FUNCTION_BLOCK OutputPipe (* Composite Function Block Type *)
  (* Standard: 61499-2 *)
  (* Version 0.0, 2011-12-23, 4DIAC-IDE, 4DIAC-Consortium *)
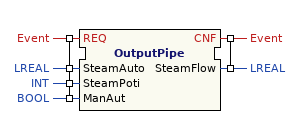
  EVENT_INPUT
    REQ WITH SteamAuto, SteamPoti, ManAut; (* Normal Execution Request *)
  END_EVENT
  EVENT_OUTPUT
    CNF WITH SteamFlow; (* Execution Confirmation *)
  END_EVENT
  VAR_INPUT
    SteamAuto : LREAL; (* Input event qualifier *)
    SteamPoti : INT;
    ManAut : BOOL; (* 0:Man, 1:Auto *)
  END_VAR
  VAR_OUTPUT
    SteamFlow : LREAL; (* Output event qualifier *)
  END_VAR
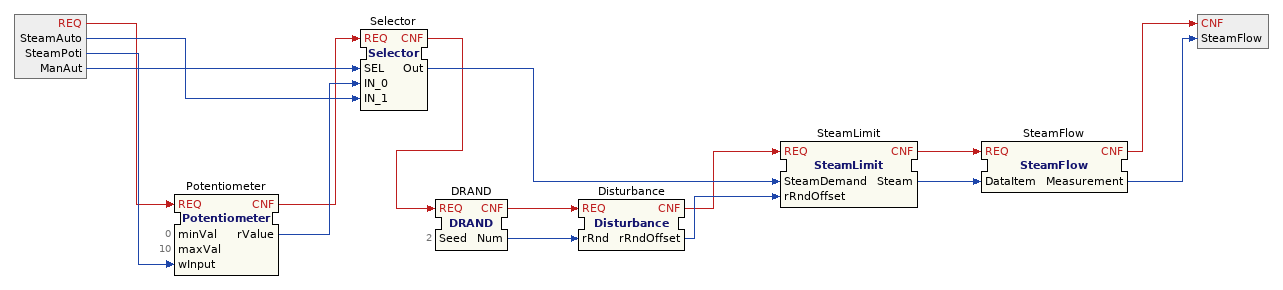
  FBS
    SteamFlow : SteamFlow;
    DRAND : DRAND(Seed := 2);
    Disturbance : Disturbance;
    SteamLimit : SteamLimit;
    Selector : Selector;
    Potentiometer : Potentiometer(minVal := 0, maxVal := 10);
  END_FBS
  EVENT_CONNECTIONS
    SteamFlow.CNF TO CNF;
    DRAND.CNF TO Disturbance.REQ;
    Disturbance.CNF TO SteamLimit.REQ;
    SteamLimit.CNF TO SteamFlow.REQ;
    Selector.CNF TO DRAND.REQ;
    REQ TO Potentiometer.REQ;
    Potentiometer.CNF TO Selector.REQ;
  END_CONNECTIONS
  DATA_CONNECTIONS
    SteamFlow.Measurement TO SteamFlow;
    DRAND.Num TO Disturbance.rRnd;
    SteamLimit.Steam TO SteamFlow.DataItem;
    Disturbance.rRndOffset TO SteamLimit.rRndOffset;
    ManAut TO Selector.SEL;
    SteamAuto TO Selector.IN_1;
    Selector.Out TO SteamLimit.SteamDemand;
    Potentiometer.rValue TO Selector.IN_0;
    SteamPoti TO Potentiometer.wInput;
  END_CONNECTIONS
END_FUNCTION_BLOCK
